# EPICS substitutions: elioApp/Db/EL1034.substitutions
file EL1034.template { pattern
{ CHAN	}
{ 1	}
{ 2	}
{ 3	}
{ 4	}
}
